FUNCTION_BLOCK DelayFeedAfterCycle (* Basic Function Block Type *)
  (* Standard: 61499-2 *)
  (* Version 0.0, 7/7/2026, Schneider Electric, Template *)
  PACKAGE SE.Nereda;
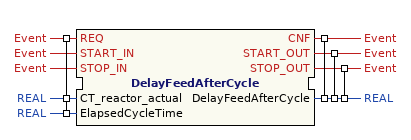
  EVENT_INPUT
    REQ WITH CT_reactor_actual, ElapsedCycleTime; (* Normal Execution Request *)
    START_IN;
    STOP_IN;
  END_EVENT
  EVENT_OUTPUT
    CNF WITH DelayFeedAfterCycle; (* Execution Confirmation *)
    START_OUT WITH DelayFeedAfterCycle;
    STOP_OUT WITH DelayFeedAfterCycle;
  END_EVENT
  VAR_INPUT
    CT_reactor_actual : REAL; (* Input event qualifier *)
    ElapsedCycleTime : REAL;
  END_VAR
  VAR_OUTPUT
    DelayFeedAfterCycle : REAL; (* Output event qualifier *)
  END_VAR
  VAR
    InDelayFeedAfterCycle : REAL;
  END_VAR
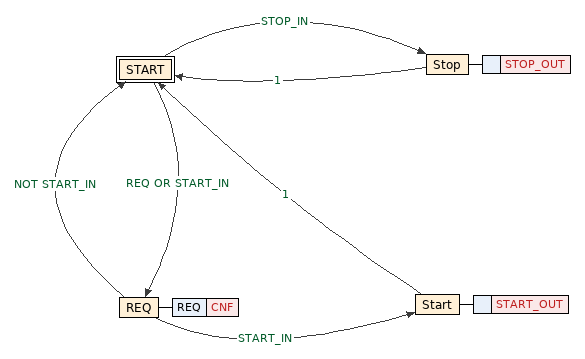
  EC_STATES
    START; (* Initial State *)
    REQ : REQ -> CNF; (* Normal execution *)
    Start : -> START_OUT;
    Stop : -> STOP_OUT;
  END_STATES
  EC_TRANSITIONS
    START TO REQ := REQ OR START_IN;
    REQ TO START := NOT START_IN;
    START TO Stop := STOP_IN;
    Stop TO START := 1;
    REQ TO Start := START_IN;
    Start TO START := 1;
  END_TRANSITIONS
  ALGORITHM REQ IN ST: (* Normally executed algorithm *)
;
InDelayFeedAfterCycle := (CT_reactor_actual - ElapsedCycleTime);

IF InDelayFeedAfterCycle > 0 THEN
	DelayFeedAfterCycle := InDelayFeedAfterCycle;
ELSE
	DelayFeedAfterCycle := 0;
END_IF;
  END_ALGORITHM
END_FUNCTION_BLOCK
